Omron CX-Programmer project NewProject (CX-Programmer 9.61)

# PLC NewPLC1: CP1E E20

## Global symbols (name address type ; comment)
0.00 BOOL  ; Push Button
0.01 BOOL  ; SystemOn
100.00 BOOL  ; M1
100.01 BOOL  ; M2
100.02 BOOL  ; M3
100.03 BOOL  ; M4
100.04 BOOL  ; M5
100.05 BOOL  ; M6
100.06 BOOL  ; M7
10.00 BOOL  ; G_P
10.01 BOOL  ; R
10.02 BOOL  ; R_P
10.03 BOOL  ; Y
10.04 BOOL  ; G
T000 BOOL  ; Timer1
T001 BOOL  ; Timer2
T002 BOOL  ; Timer3
T003 BOOL  ; Timer4
T004 BOOL  ; Timer5
T005 BOOL  ; Timer6
T006 BOOL  ; Timer7

## Program NewProgram1 (cyclic task 0)

### Section Section1

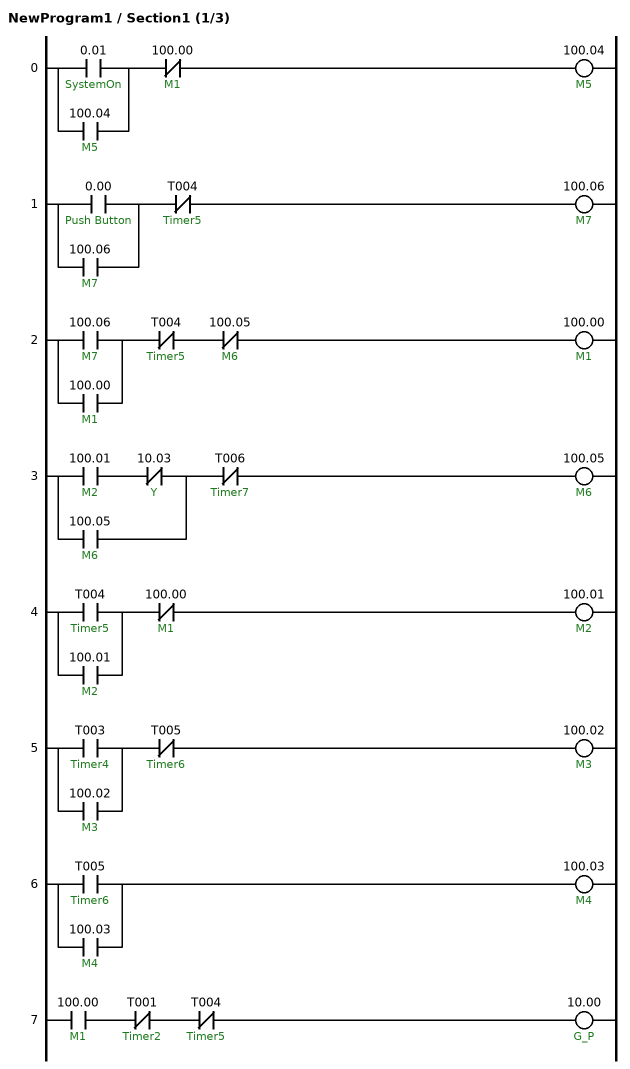
; rung 0
LD 0.01  ; SystemOn
OR 100.04  ; M5
ANDNOT 100.00  ; M1
OUT 100.04  ; M5
; rung 1
LD 0.00  ; Push Button
OR 100.06  ; M7
ANDNOT T004  ; Timer5
OUT 100.06  ; M7
; rung 2
LD 100.06  ; M7
OR 100.00  ; M1
ANDNOT T004  ; Timer5
ANDNOT 100.05  ; M6
OUT 100.00  ; M1
; rung 3
LD 100.01  ; M2
ANDNOT 10.03  ; Y
OR 100.05  ; M6
ANDNOT T006  ; Timer7
OUT 100.05  ; M6
; rung 4
LD T004  ; Timer5
OR 100.01  ; M2
ANDNOT 100.00  ; M1
OUT 100.01  ; M2
; rung 5
LD T003  ; Timer4
OR 100.02  ; M3
ANDNOT T005  ; Timer6
OUT 100.02  ; M3
; rung 6
LD T005  ; Timer6
OR 100.03  ; M4
OUT 100.03  ; M4
; rung 7
LD 100.00  ; M1
ANDNOT T001  ; Timer2
ANDNOT T004  ; Timer5
OUT 10.00  ; G_P

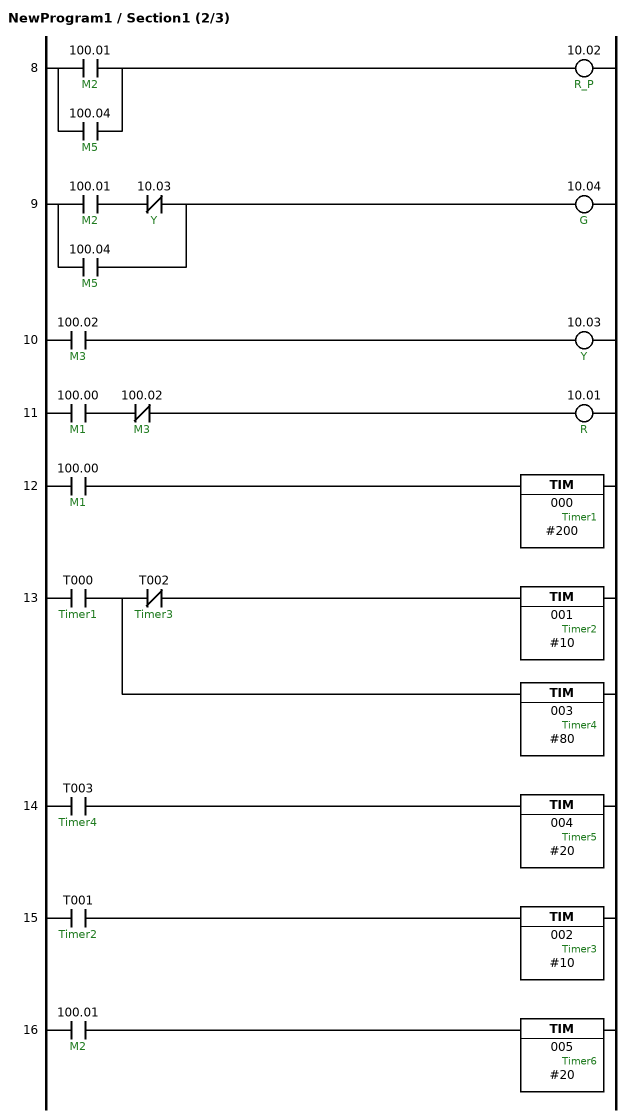
; rung 8
LD 100.01  ; M2
OR 100.04  ; M5
OUT 10.02  ; R_P
; rung 9
LD 100.01  ; M2
ANDNOT 10.03  ; Y
OR 100.04  ; M5
OUT 10.04  ; G
; rung 10
LD 100.02  ; M3
OUT 10.03  ; Y
; rung 11
LD 100.00  ; M1
ANDNOT 100.02  ; M3
OUT 10.01  ; R
; rung 12
LD 100.00  ; M1
TIM 000 #200  ; Timer1
; rung 13
LD T000  ; Timer1
OUT TR0
ANDNOT T002  ; Timer3
TIM 001 #10  ; Timer2
LD TR0
TIM 003 #80  ; Timer4
; rung 14
LD T003  ; Timer4
TIM 004 #20  ; Timer5
; rung 15
LD T001  ; Timer2
TIM 002 #10  ; Timer3
; rung 16
LD 100.01  ; M2
TIM 005 #20  ; Timer6

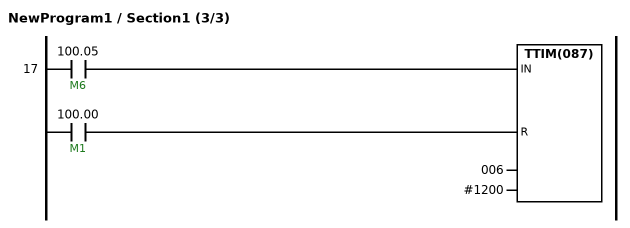
; rung 17
LD 100.05  ; M6
LD 100.00  ; M1
TTIM(087) 006 #1200  ; Timer7

### Section END
; rung 0
END(001)